FUNCTION_BLOCK MovingStatus (* Basic Function Block Type *)
  (* Standard: 61499-2 *)
  (* Version 0.0, 12/5/2011, XPMUser, nxtControl GmbH, Template *)
  PACKAGE Main;
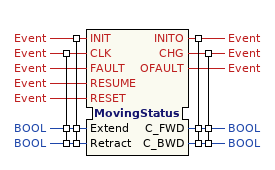
  EVENT_INPUT
    INIT WITH Extend, Retract; (* Initialization Request *)
    CLK WITH Extend, Retract; (* Clock signal *)
    FAULT;
    RESUME;
    RESET;
  END_EVENT
  EVENT_OUTPUT
    INITO WITH C_FWD, C_BWD; (* Initialization Confirm *)
    CHG WITH C_FWD, C_BWD; (* Data outputs changed *)
    OFAULT;
  END_EVENT
  VAR_INPUT
    Extend : BOOL; (* Move forwards *)
    Retract : BOOL; (* Move backwards *)
  END_VAR
  VAR_OUTPUT
    C_FWD : BOOL; (* Confirmed move forwards *)
    C_BWD : BOOL; (* Confirmed move backwards *)
  END_VAR
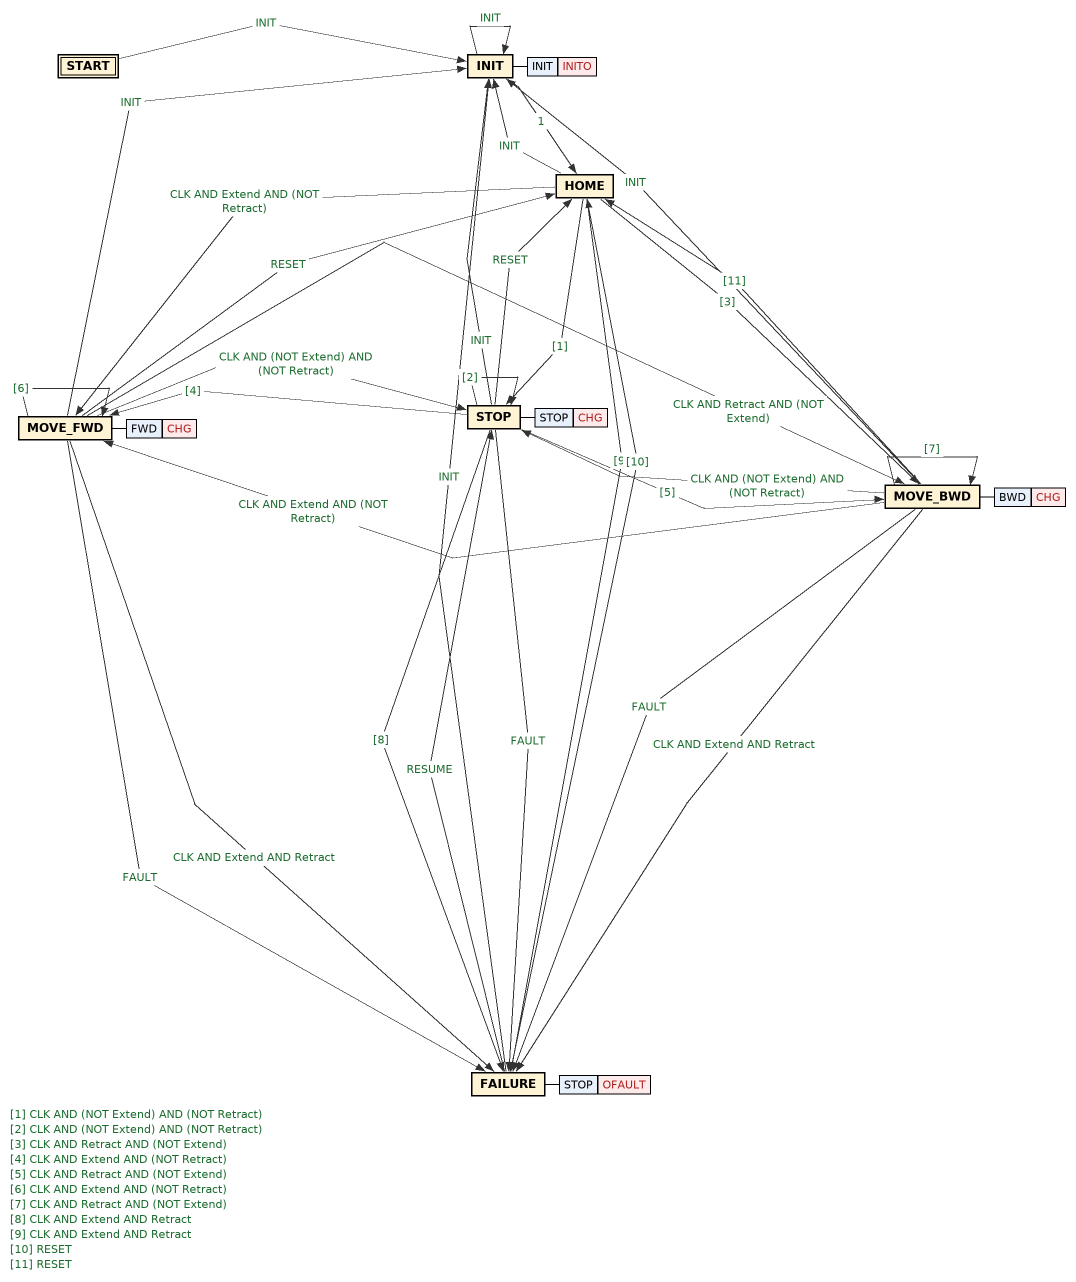
  EC_STATES
    START; (* Initial State *)
    INIT : INIT -> INITO; (* Initialization *)
    MOVE_FWD : FWD -> CHG;
    MOVE_BWD : BWD -> CHG;
    STOP : STOP -> CHG;
    FAILURE : STOP -> OFAULT;
    HOME;
  END_STATES
  EC_TRANSITIONS
    START TO INIT := INIT;
    HOME TO MOVE_FWD := CLK AND Extend AND (NOT Retract);
    HOME TO STOP := CLK AND (NOT Extend) AND (NOT Retract);
    HOME TO MOVE_BWD := CLK AND Retract AND (NOT Extend);
    MOVE_FWD TO FAILURE := FAULT;
    STOP TO FAILURE := FAULT;
    MOVE_BWD TO FAILURE := FAULT;
    MOVE_FWD TO STOP := CLK AND (NOT Extend) AND (NOT Retract);
    MOVE_BWD TO STOP := CLK AND (NOT Extend) AND (NOT Retract);
    STOP TO MOVE_FWD := CLK AND Extend AND (NOT Retract);
    STOP TO MOVE_BWD := CLK AND Retract AND (NOT Extend);
    FAILURE TO STOP := RESUME;
    MOVE_FWD TO MOVE_BWD := CLK AND Retract AND (NOT Extend);
    MOVE_BWD TO MOVE_FWD := CLK AND Extend AND (NOT Retract);
    STOP TO FAILURE := CLK AND Extend AND Retract;
    HOME TO FAILURE := CLK AND Extend AND Retract;
    MOVE_FWD TO FAILURE := CLK AND Extend AND Retract;
    MOVE_BWD TO FAILURE := CLK AND Extend AND Retract;
    MOVE_FWD TO MOVE_FWD := CLK AND Extend AND (NOT Retract);
    MOVE_BWD TO MOVE_BWD := CLK AND Retract AND (NOT Extend);
    STOP TO STOP := CLK AND (NOT Extend) AND (NOT Retract);
    MOVE_BWD TO INIT := INIT;
    MOVE_FWD TO INIT := INIT;
    STOP TO INIT := INIT;
    FAILURE TO INIT := INIT;
    INIT TO INIT := INIT;
    FAILURE TO HOME := RESET;
    MOVE_BWD TO HOME := RESET;
    MOVE_FWD TO HOME := RESET;
    INIT TO HOME := 1;
    STOP TO HOME := RESET;
    HOME TO INIT := INIT;
  END_TRANSITIONS
  ALGORITHM INIT IN ST: (* Initialization algorithm *)
INIT:=FALSE;
C_FWD := FALSE;
C_BWD := FALSE;
  END_ALGORITHM
  ALGORITHM FWD IN ST: (* Normally executed algorithm *)
CLK:=FALSE;
C_FWD := TRUE;
C_BWD := FALSE;
  END_ALGORITHM
  ALGORITHM BWD IN ST:
CLK := FALSE;
C_FWD := FALSE;
C_BWD := TRUE;
  END_ALGORITHM
  ALGORITHM STOP IN ST:
CLK := FALSE;
C_FWD := FALSE;
C_BWD := FALSE;
  END_ALGORITHM
END_FUNCTION_BLOCK
